// TIA Portal V19 export
FUNCTION_BLOCK "Decoiler_PneumaticBrake"   // FB26, LAD
TITLE = DECOILER PNEUMATIC BRAKE
// stored: MemoryReserve 100, SetENOAutomatically false
   VAR_INPUT
      AreaInterface : "AreaInterface";
      PbOpenClose : Bool;
      PbPartilaOpenClose : Bool;
      Open_Req_FeedMotor : Bool;
      Open_Req_Snubber : Bool;
      Partial_Req : Bool;
      InLine : Bool;
      DiameterValue : Real;
   END_VAR
   VAR_OUTPUT
      Open : Bool;
      Lamp_Open_Forced : Bool;
      Lamp_Partial_Forced : Bool;
      V_Open : Bool;
      V_PartialHigh : Bool;
      V_PartialLow : Bool;
   END_VAR
   VAR_IN_OUT
      PersistentValues : "Decoiler_Pers";
   END_VAR
   VAR
      Sts : Struct
         IsOpen : Bool;
         Open_Req_Pb : Bool;
         Partial_Req_Pb : Bool;
      END_STRUCT;
      Ctrl : Struct
         Open : Bool;
         Partial : Bool;
      END_STRUCT;
      Aux_PbOpenClose : Bool;
      TON_BrakeisOpen : IEC_TIMER;
   END_VAR
   VAR_TEMP
      Set : Bool;
      Rst : Bool;
   END_VAR
   VAR_TEMP   // added for the SCL form of the ladder/FBD networks
      _w1 : Bool;
   END_VAR
BEGIN

REGION Network 1: Total open
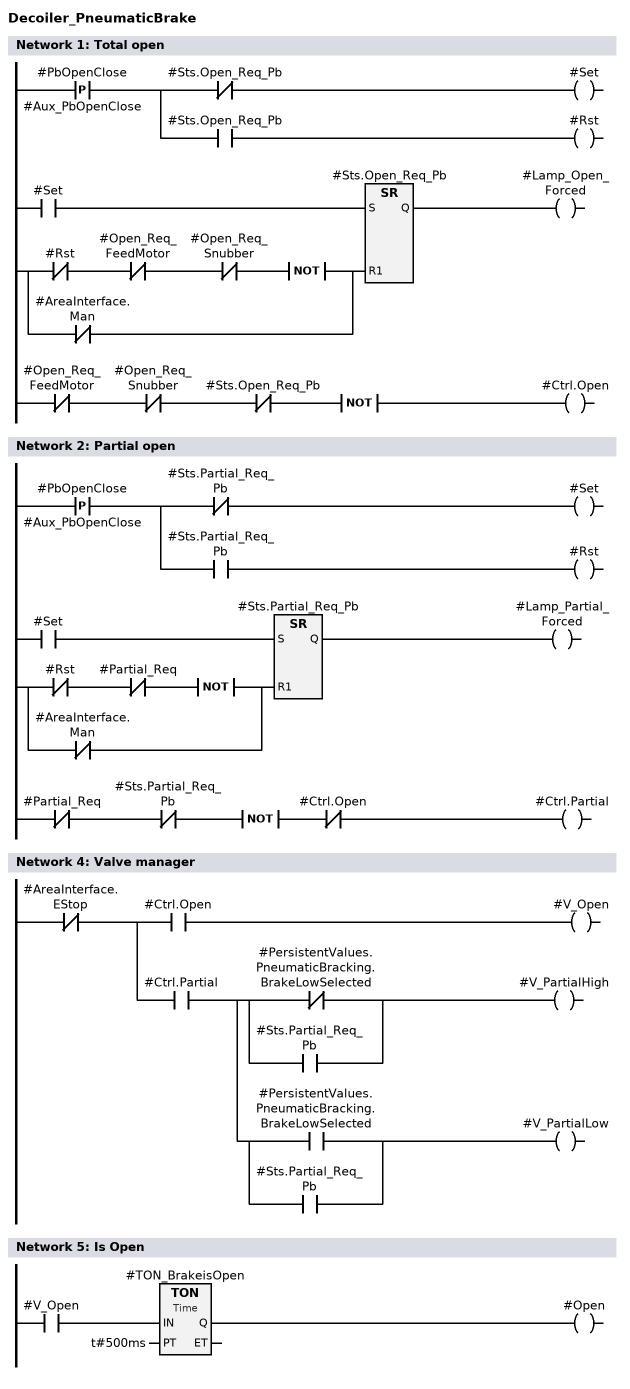
   RUNG wire#powerrail
      P_Contact(operand := #PbOpenClose, bit := #Aux_PbOpenClose)
      wire#w1
      I_Contact( #Sts.Open_Req_Pb )
      Coil( #Set )
   END_RUNG
   RUNG wire#w1
      Contact( #Sts.Open_Req_Pb )
      Coil( #Rst )
   END_RUNG
   RUNG wire#powerrail
      Contact( #Set )
      S_SR(operand := #Sts.Open_Req_Pb, r1 := wire#w2)
      Coil( #Lamp_Open_Forced )
   END_RUNG
   RUNG wire#powerrail
      I_Contact( #Rst )
      I_Contact( #Open_Req_FeedMotor )
      I_Contact( #Open_Req_Snubber )
      Not()
   END_RUNG wire#w2
   RUNG wire#powerrail
      I_Contact( #AreaInterface.Man )
   END_RUNG wire#w2
   RUNG wire#powerrail
      I_Contact( #Open_Req_FeedMotor )
      I_Contact( #Open_Req_Snubber )
      I_Contact( #Sts.Open_Req_Pb )
      Not()
      Coil( #Ctrl.Open )
   END_RUNG
   // the same network as SCL:
   #_w1 := #PbOpenClose AND NOT #Aux_PbOpenClose;   // rising edge of #PbOpenClose
   #Aux_PbOpenClose := #PbOpenClose;
   #Set := #_w1 AND NOT #Sts.Open_Req_Pb;
   #Rst := #_w1 AND #Sts.Open_Req_Pb;
   IF #Set THEN
       #Sts.Open_Req_Pb := TRUE;   // SR flip-flop
   END_IF;
   IF NOT (NOT #Rst AND NOT #Open_Req_FeedMotor AND NOT #Open_Req_Snubber) OR NOT #AreaInterface.Man THEN
       #Sts.Open_Req_Pb := FALSE;
   END_IF;
   #Lamp_Open_Forced := #Sts.Open_Req_Pb;
   #Ctrl.Open := NOT (NOT #Open_Req_FeedMotor AND NOT #Open_Req_Snubber AND NOT #Sts.Open_Req_Pb);
END_REGION

REGION Network 2: Partial open
   RUNG wire#powerrail
      P_Contact(operand := #PbOpenClose, bit := #Aux_PbOpenClose)
      wire#w1
      I_Contact( #Sts.Partial_Req_Pb )
      Coil( #Set )
   END_RUNG
   RUNG wire#w1
      Contact( #Sts.Partial_Req_Pb )
      Coil( #Rst )
   END_RUNG
   RUNG wire#powerrail
      Contact( #Set )
      S_SR(operand := #Sts.Partial_Req_Pb, r1 := wire#w2)
      Coil( #Lamp_Partial_Forced )
   END_RUNG
   RUNG wire#powerrail
      I_Contact( #Rst )
      I_Contact( #Partial_Req )
      Not()
   END_RUNG wire#w2
   RUNG wire#powerrail
      I_Contact( #AreaInterface.Man )
   END_RUNG wire#w2
   RUNG wire#powerrail
      I_Contact( #Partial_Req )
      I_Contact( #Sts.Partial_Req_Pb )
      Not()
      I_Contact( #Ctrl.Open )
      Coil( #Ctrl.Partial )
   END_RUNG
   // the same network as SCL:
   #_w1 := #PbOpenClose AND NOT #Aux_PbOpenClose;   // rising edge of #PbOpenClose
   #Aux_PbOpenClose := #PbOpenClose;
   #Set := #_w1 AND NOT #Sts.Partial_Req_Pb;
   #Rst := #_w1 AND #Sts.Partial_Req_Pb;
   IF #Set THEN
       #Sts.Partial_Req_Pb := TRUE;   // SR flip-flop
   END_IF;
   IF NOT (NOT #Rst AND NOT #Partial_Req) OR NOT #AreaInterface.Man THEN
       #Sts.Partial_Req_Pb := FALSE;
   END_IF;
   #Lamp_Partial_Forced := #Sts.Partial_Req_Pb;
   #Ctrl.Partial := NOT (NOT #Partial_Req AND NOT #Sts.Partial_Req_Pb) AND NOT #Ctrl.Open;
END_REGION

REGION Network 3 (SCL): Partial brake with diameter

   IF #InLine AND #PersistentValues.CoilDiamSensor.Par.AnalogicSensor_Enable THEN

       IF #Ctrl.Partial AND
           #DiameterValue < #PersistentValues.PneumaticBracking.DiameterChangeBrake
       THEN

           #PersistentValues.PneumaticBracking.BrakeLowSelected := TRUE;
       END_IF;

   ELSE

       #PersistentValues.PneumaticBracking.BrakeLowSelected := FALSE;

   END_IF;
END_REGION

REGION Network 4: Valve manager
   RUNG wire#powerrail
      I_Contact( #AreaInterface.EStop )
      wire#w1
      Contact( #Ctrl.Open )
      Coil( #V_Open )
   END_RUNG
   RUNG wire#w1
      Contact( #Ctrl.Partial )
      wire#w2
      I_Contact( #PersistentValues.PneumaticBracking.BrakeLowSelected )
      wire#w3
      Coil( #V_PartialHigh )
   END_RUNG
   RUNG wire#w2
      Contact( #Sts.Partial_Req_Pb )
   END_RUNG wire#w3
   RUNG wire#w2
      Contact( #PersistentValues.PneumaticBracking.BrakeLowSelected )
      wire#w4
      Coil( #V_PartialLow )
   END_RUNG
   RUNG wire#w2
      Contact( #Sts.Partial_Req_Pb )
   END_RUNG wire#w4
   // the same network as SCL:
   #V_Open := NOT #AreaInterface.EStop AND #Ctrl.Open;
   #_w1 := NOT #AreaInterface.EStop AND #Ctrl.Partial;
   #V_PartialHigh := #_w1 AND (NOT #PersistentValues.PneumaticBracking.BrakeLowSelected OR #Sts.Partial_Req_Pb);
   #V_PartialLow := #_w1 AND (#PersistentValues.PneumaticBracking.BrakeLowSelected OR #Sts.Partial_Req_Pb);
END_REGION

REGION Network 5: Is Open
   RUNG wire#powerrail
      Contact( #V_Open )
      { S7_Templates := "time_type := Time" } #TON_BrakeisOpen.TON(pt := t#500ms, et =>)
      Coil( #Open )
   END_RUNG
   // the same network as SCL:
   #TON_BrakeisOpen.TON(IN := #V_Open, PT := t#500ms);
   #Open := #TON_BrakeisOpen.Q;
END_REGION
END_FUNCTION_BLOCK
